   1:  PR[GP1:91,1] = PR[GP1:90,1] + 133.078;
   1:  PR[GP1:91,2] = PR[GP1:90,2] + 104.334;
   1:L PR[91] 10mm/sec FINE;
   1:  PR[GP1:91,1] = PR[GP1:90,1] + 132.574;
   1:  PR[GP1:91,2] = PR[GP1:90,2] + 104.937;
   1:L PR[91] 10mm/sec FINE;
   1:  PR[GP1:91,1] = PR[GP1:90,1] + 131.283;
   1:  PR[GP1:91,2] = PR[GP1:90,2] + 106.321;
   1:L PR[91] 10mm/sec FINE;
   1:  PR[GP1:91,1] = PR[GP1:90,1] + 130.348;
   1:  PR[GP1:91,2] = PR[GP1:90,2] + 107.265;
   1:L PR[91] 10mm/sec FINE;
   1:  PR[GP1:91,1] = PR[GP1:90,1] + 129.842;
   1:  PR[GP1:91,2] = PR[GP1:90,2] + 107.719;
   1:L PR[91] 10mm/sec FINE;
   1:  PR[GP1:91,1] = PR[GP1:90,1] + 128.720;
   1:  PR[GP1:91,2] = PR[GP1:90,2] + 108.706;
   1:L PR[91] 10mm/sec FINE;
   1:  PR[GP1:91,1] = PR[GP1:90,1] + 125.281;
   1:  PR[GP1:91,2] = PR[GP1:90,2] + 111.248;
   1:L PR[91] 10mm/sec FINE;
   1:  PR[GP1:91,1] = PR[GP1:90,1] + 124.815;
   1:  PR[GP1:91,2] = PR[GP1:90,2] + 111.519;
   1:L PR[91] 10mm/sec FINE;
   1:  PR[GP1:91,1] = PR[GP1:90,1] + 123.935;
   1:  PR[GP1:91,2] = PR[GP1:90,2] + 111.995;
   1:L PR[91] 10mm/sec FINE;
   1:  PR[GP1:91,1] = PR[GP1:90,1] + 122.852;
   1:  PR[GP1:91,2] = PR[GP1:90,2] + 112.673;
   1:L PR[91] 10mm/sec FINE;
   1:  PR[GP1:91,1] = PR[GP1:90,1] + 122.591;
   1:  PR[GP1:91,2] = PR[GP1:90,2] + 112.818;
   1:L PR[91] 10mm/sec FINE;
   1:  PR[GP1:91,1] = PR[GP1:90,1] + 122.383;
   1:  PR[GP1:91,2] = PR[GP1:90,2] + 112.910;
   1:L PR[91] 10mm/sec FINE;
   1:  PR[GP1:91,1] = PR[GP1:90,1] + 121.910;
   1:  PR[GP1:91,2] = PR[GP1:90,2] + 113.234;
   1:L PR[91] 10mm/sec FINE;
   1:  PR[GP1:91,1] = PR[GP1:90,1] + 120.972;
   1:  PR[GP1:91,2] = PR[GP1:90,2] + 113.697;
   1:L PR[91] 10mm/sec FINE;
   1:  PR[GP1:91,1] = PR[GP1:90,1] + 120.433;
   1:  PR[GP1:91,2] = PR[GP1:90,2] + 113.889;
   1:L PR[91] 10mm/sec FINE;
   1:  PR[GP1:91,1] = PR[GP1:90,1] + 118.110;
   1:  PR[GP1:91,2] = PR[GP1:90,2] + 115.002;
   1:L PR[91] 10mm/sec FINE;
   1:  PR[GP1:91,1] = PR[GP1:90,1] + 115.533;
   1:  PR[GP1:91,2] = PR[GP1:90,2] + 115.758;
   1:L PR[91] 10mm/sec FINE;
   1:  PR[GP1:91,1] = PR[GP1:90,1] + 114.209;
   1:  PR[GP1:91,2] = PR[GP1:90,2] + 116.169;
   1:L PR[91] 10mm/sec FINE;
   1:  PR[GP1:91,1] = PR[GP1:90,1] + 112.597;
   1:  PR[GP1:91,2] = PR[GP1:90,2] + 116.362;
   1:L PR[91] 10mm/sec FINE;
   1:  PR[GP1:91,1] = PR[GP1:90,1] + 110.291;
   1:  PR[GP1:91,2] = PR[GP1:90,2] + 116.663;
   1:L PR[91] 10mm/sec FINE;
   1:  PR[GP1:91,1] = PR[GP1:90,1] + 108.430;
   1:  PR[GP1:91,2] = PR[GP1:90,2] + 116.678;
   1:L PR[91] 10mm/sec FINE;
   1:  PR[GP1:91,1] = PR[GP1:90,1] + 104.683;
   1:  PR[GP1:91,2] = PR[GP1:90,2] + 116.533;
   1:L PR[91] 10mm/sec FINE;
   1:  PR[GP1:91,1] = PR[GP1:90,1] + 104.119;
   1:  PR[GP1:91,2] = PR[GP1:90,2] + 116.445;
   1:L PR[91] 10mm/sec FINE;
   1:  PR[GP1:91,1] = PR[GP1:90,1] + 100.824;
   1:  PR[GP1:91,2] = PR[GP1:90,2] + 115.784;
   1:L PR[91] 10mm/sec FINE;
   1:  PR[GP1:91,1] = PR[GP1:90,1] + 99.441;
   1:  PR[GP1:91,2] = PR[GP1:90,2] + 115.278;
   1:L PR[91] 10mm/sec FINE;
   1:  PR[GP1:91,1] = PR[GP1:90,1] + 97.150;
   1:  PR[GP1:91,2] = PR[GP1:90,2] + 114.379;
   1:L PR[91] 10mm/sec FINE;
   1:  PR[GP1:91,1] = PR[GP1:90,1] + 96.875;
   1:  PR[GP1:91,2] = PR[GP1:90,2] + 114.236;
   1:L PR[91] 10mm/sec FINE;
   1:  PR[GP1:91,1] = PR[GP1:90,1] + 94.091;
   1:  PR[GP1:91,2] = PR[GP1:90,2] + 112.451;
   1:L PR[91] 10mm/sec FINE;
   1:  PR[GP1:91,1] = PR[GP1:90,1] + 93.175;
   1:  PR[GP1:91,2] = PR[GP1:90,2] + 111.645;
   1:L PR[91] 10mm/sec FINE;
   1:  PR[GP1:91,1] = PR[GP1:90,1] + 91.727;
   1:  PR[GP1:91,2] = PR[GP1:90,2] + 110.082;
   1:L PR[91] 10mm/sec FINE;
   1:  PR[GP1:91,1] = PR[GP1:90,1] + 91.060;
   1:  PR[GP1:91,2] = PR[GP1:90,2] + 109.259;
   1:L PR[91] 10mm/sec FINE;
   1:  PR[GP1:91,1] = PR[GP1:90,1] + 90.553;
   1:  PR[GP1:91,2] = PR[GP1:90,2] + 108.353;
   1:L PR[91] 10mm/sec FINE;
   1:  PR[GP1:91,1] = PR[GP1:90,1] + 89.537;
   1:  PR[GP1:91,2] = PR[GP1:90,2] + 106.416;
   1:L PR[91] 10mm/sec FINE;
   1:  PR[GP1:91,1] = PR[GP1:90,1] + 89.209;
   1:  PR[GP1:91,2] = PR[GP1:90,2] + 105.500;
   1:L PR[91] 10mm/sec FINE;
   1:  PR[GP1:91,1] = PR[GP1:90,1] + 88.715;
   1:  PR[GP1:91,2] = PR[GP1:90,2] + 103.374;
   1:L PR[91] 10mm/sec FINE;
   1:  PR[GP1:91,1] = PR[GP1:90,1] + 88.529;
   1:  PR[GP1:91,2] = PR[GP1:90,2] + 102.358;
   1:L PR[91] 10mm/sec FINE;
   1:  PR[GP1:91,1] = PR[GP1:90,1] + 88.508;
   1:  PR[GP1:91,2] = PR[GP1:90,2] + 101.310;
   1:L PR[91] 10mm/sec FINE;
   1:  PR[GP1:91,1] = PR[GP1:90,1] + 88.621;
   1:  PR[GP1:91,2] = PR[GP1:90,2] + 99.170;
   1:L PR[91] 10mm/sec FINE;
   1:  PR[GP1:91,1] = PR[GP1:90,1] + 88.809;
   1:  PR[GP1:91,2] = PR[GP1:90,2] + 98.011;
   1:L PR[91] 10mm/sec FINE;
   1:  PR[GP1:91,1] = PR[GP1:90,1] + 88.822;
   1:  PR[GP1:91,2] = PR[GP1:90,2] + 97.961;
   1:L PR[91] 10mm/sec FINE;
   1:  PR[GP1:91,1] = PR[GP1:90,1] + 89.980;
   1:  PR[GP1:91,2] = PR[GP1:90,2] + 94.456;
   1:L PR[91] 10mm/sec FINE;
   1:  PR[GP1:91,1] = PR[GP1:90,1] + 90.236;
   1:  PR[GP1:91,2] = PR[GP1:90,2] + 93.612;
   1:L PR[91] 10mm/sec FINE;
   1:  PR[GP1:91,1] = PR[GP1:90,1] + 91.520;
   1:  PR[GP1:91,2] = PR[GP1:90,2] + 92.149;
   1:  PR[GP1:91,3] = PR[GP1:90,3] + 65.900;
   1:L PR[91] 10mm/sec FINE;
   1:  PR[GP1:91,1] = PR[GP1:90,1] + 92.735;
   1:  PR[GP1:91,2] = PR[GP1:90,2] + 90.111;
   1:L PR[91] 10mm/sec FINE;
   1:  PR[GP1:91,1] = PR[GP1:90,1] + 95.040;
   1:  PR[GP1:91,2] = PR[GP1:90,2] + 86.918;
   1:L PR[91] 10mm/sec FINE;
   1:  PR[GP1:91,1] = PR[GP1:90,1] + 96.371;
   1:  PR[GP1:91,2] = PR[GP1:90,2] + 85.475;
   1:L PR[91] 10mm/sec FINE;
   1:  PR[GP1:91,1] = PR[GP1:90,1] + 97.440;
   1:  PR[GP1:91,2] = PR[GP1:90,2] + 84.369;
   1:L PR[91] 10mm/sec FINE;
   1:  PR[GP1:91,1] = PR[GP1:90,1] + 101.784;
   1:  PR[GP1:91,2] = PR[GP1:90,2] + 80.978;
   1:L PR[91] 10mm/sec FINE;
   1:  PR[GP1:91,1] = PR[GP1:90,1] + 102.201;
   1:  PR[GP1:91,2] = PR[GP1:90,2] + 80.753;
   1:L PR[91] 10mm/sec FINE;
   1:  PR[GP1:91,1] = PR[GP1:90,1] + 106.860;
   1:  PR[GP1:91,2] = PR[GP1:90,2] + 78.023;
   1:L PR[91] 10mm/sec FINE;
   1:  PR[GP1:91,1] = PR[GP1:90,1] + 113.422;
   1:  PR[GP1:91,2] = PR[GP1:90,2] + 75.517;
   1:L PR[91] 10mm/sec FINE;
   1:  PR[GP1:91,1] = PR[GP1:90,1] + 117.856;
   1:  PR[GP1:91,2] = PR[GP1:90,2] + 74.650;
   1:L PR[91] 10mm/sec FINE;
   1:  PR[GP1:91,1] = PR[GP1:90,1] + 120.560;
   1:  PR[GP1:91,2] = PR[GP1:90,2] + 74.494;
   1:L PR[91] 10mm/sec FINE;
   1:  PR[GP1:91,1] = PR[GP1:90,1] + 121.439;
   1:  PR[GP1:91,2] = PR[GP1:90,2] + 74.463;
   1:L PR[91] 10mm/sec FINE;
   1:  PR[GP1:91,1] = PR[GP1:90,1] + 123.315;
   1:  PR[GP1:91,2] = PR[GP1:90,2] + 74.706;
   1:L PR[91] 10mm/sec FINE;
   1:  PR[GP1:91,1] = PR[GP1:90,1] + 125.689;
   1:  PR[GP1:91,2] = PR[GP1:90,2] + 74.966;
   1:L PR[91] 10mm/sec FINE;
   1:  PR[GP1:91,1] = PR[GP1:90,1] + 127.460;
   1:  PR[GP1:91,2] = PR[GP1:90,2] + 75.437;
   1:L PR[91] 10mm/sec FINE;
   1:  PR[GP1:91,1] = PR[GP1:90,1] + 130.068;
   1:  PR[GP1:91,2] = PR[GP1:90,2] + 76.445;
   1:L PR[91] 10mm/sec FINE;
   1:  PR[GP1:91,1] = PR[GP1:90,1] + 131.522;
   1:  PR[GP1:91,2] = PR[GP1:90,2] + 77.116;
   1:L PR[91] 10mm/sec FINE;
   1:  PR[GP1:91,1] = PR[GP1:90,1] + 132.509;
   1:  PR[GP1:91,2] = PR[GP1:90,2] + 77.819;
   1:L PR[91] 10mm/sec FINE;
   1:  PR[GP1:91,1] = PR[GP1:90,1] + 134.897;
   1:  PR[GP1:91,2] = PR[GP1:90,2] + 79.695;
   1:L PR[91] 10mm/sec FINE;
   1:  PR[GP1:91,1] = PR[GP1:90,1] + 135.682;
   1:  PR[GP1:91,2] = PR[GP1:90,2] + 80.533;
   1:L PR[91] 10mm/sec FINE;
   1:  PR[GP1:91,1] = PR[GP1:90,1] + 137.230;
   1:  PR[GP1:91,2] = PR[GP1:90,2] + 82.841;
   1:L PR[91] 10mm/sec FINE;
   1:  PR[GP1:91,1] = PR[GP1:90,1] + 137.802;
   1:  PR[GP1:91,2] = PR[GP1:90,2] + 83.791;
   1:L PR[91] 10mm/sec FINE;
   1:  PR[GP1:91,1] = PR[GP1:90,1] + 138.178;
   1:  PR[GP1:91,2] = PR[GP1:90,2] + 84.884;
   1:L PR[91] 10mm/sec FINE;
   1:  PR[GP1:91,1] = PR[GP1:90,1] + 138.856;
   1:  PR[GP1:91,2] = PR[GP1:90,2] + 86.970;
   1:L PR[91] 10mm/sec FINE;
   1:  PR[GP1:91,1] = PR[GP1:90,1] + 139.017;
   1:  PR[GP1:91,2] = PR[GP1:90,2] + 88.230;
   1:L PR[91] 10mm/sec FINE;
   1:  PR[GP1:91,1] = PR[GP1:90,1] + 139.191;
   1:  PR[GP1:91,2] = PR[GP1:90,2] + 90.045;
   1:L PR[91] 10mm/sec FINE;
   1:  PR[GP1:91,1] = PR[GP1:90,1] + 139.096;
   1:  PR[GP1:91,2] = PR[GP1:90,2] + 91.544;
   1:L PR[91] 10mm/sec FINE;
   1:  PR[GP1:91,1] = PR[GP1:90,1] + 138.958;
   1:  PR[GP1:91,2] = PR[GP1:90,2] + 93.171;
   1:L PR[91] 10mm/sec FINE;
   1:  PR[GP1:91,1] = PR[GP1:90,1] + 138.190;
   1:  PR[GP1:91,2] = PR[GP1:90,2] + 96.327;
   1:L PR[91] 10mm/sec FINE;
   1:  PR[GP1:91,1] = PR[GP1:90,1] + 137.095;
   1:  PR[GP1:91,2] = PR[GP1:90,2] + 99.086;
   1:L PR[91] 10mm/sec FINE;
   1:  PR[GP1:91,1] = PR[GP1:90,1] + 135.819;
   1:  PR[GP1:91,2] = PR[GP1:90,2] + 101.448;
   1:L PR[91] 10mm/sec FINE;
   1:  PR[GP1:91,1] = PR[GP1:90,1] + 135.643;
   1:  PR[GP1:91,2] = PR[GP1:90,2] + 101.737;
   1:L PR[91] 10mm/sec FINE;
   1:  PR[GP1:91,1] = PR[GP1:90,1] + 133.904;
   1:  PR[GP1:91,2] = PR[GP1:90,2] + 104.039;
   1:L PR[91] 10mm/sec FINE;
   1:  PR[GP1:91,1] = PR[GP1:90,1] + 133.599;
   1:  PR[GP1:91,2] = PR[GP1:90,2] + 104.403;
   1:L PR[91] 10mm/sec FINE;
   1:  PR[GP1:91,1] = PR[GP1:90,1] + 132.037;
   1:  PR[GP1:91,2] = PR[GP1:90,2] + 106.078;
   1:L PR[91] 10mm/sec FINE;
   1:  PR[GP1:91,1] = PR[GP1:90,1] + 131.332;
   1:  PR[GP1:91,2] = PR[GP1:90,2] + 106.790;
   1:L PR[91] 10mm/sec FINE;
   1:  PR[GP1:91,1] = PR[GP1:90,1] + 129.467;
   1:  PR[GP1:91,2] = PR[GP1:90,2] + 108.438;
   1:L PR[91] 10mm/sec FINE;
   1:  PR[GP1:91,1] = PR[GP1:90,1] + 127.205;
   1:  PR[GP1:91,2] = PR[GP1:90,2] + 110.116;
   1:L PR[91] 10mm/sec FINE;
   1:  PR[GP1:91,1] = PR[GP1:90,1] + 126.171;
   1:  PR[GP1:91,2] = PR[GP1:90,2] + 110.860;
   1:L PR[91] 10mm/sec FINE;
   1:  PR[GP1:91,1] = PR[GP1:90,1] + 125.079;
   1:  PR[GP1:91,2] = PR[GP1:90,2] + 111.497;
   1:L PR[91] 10mm/sec FINE;
   1:  PR[GP1:91,1] = PR[GP1:90,1] + 123.052;
   1:  PR[GP1:91,2] = PR[GP1:90,2] + 112.592;
   1:L PR[91] 10mm/sec FINE;
   1:  PR[GP1:91,1] = PR[GP1:90,1] + 122.515;
   1:  PR[GP1:91,2] = PR[GP1:90,2] + 112.928;
   1:L PR[91] 10mm/sec FINE;
   1:  PR[GP1:91,1] = PR[GP1:90,1] + 121.714;
   1:  PR[GP1:91,2] = PR[GP1:90,2] + 113.284;
   1:L PR[91] 10mm/sec FINE;
   1:  PR[GP1:91,1] = PR[GP1:90,1] + 120.818;
   1:  PR[GP1:91,2] = PR[GP1:90,2] + 113.730;
   1:L PR[91] 10mm/sec FINE;
   1:  PR[GP1:91,1] = PR[GP1:90,1] + 119.914;
   1:  PR[GP1:91,2] = PR[GP1:90,2] + 114.053;
   1:L PR[91] 10mm/sec FINE;
   1:  PR[GP1:91,1] = PR[GP1:90,1] + 118.581;
   1:  PR[GP1:91,2] = PR[GP1:90,2] + 114.689;
   1:L PR[91] 10mm/sec FINE;
   1:  PR[GP1:91,1] = PR[GP1:90,1] + 118.083;
   1:  PR[GP1:91,2] = PR[GP1:90,2] + 114.849;
   1:L PR[91] 10mm/sec FINE;
   1:  PR[GP1:91,1] = PR[GP1:90,1] + 117.577;
   1:  PR[GP1:91,2] = PR[GP1:90,2] + 114.961;
   1:L PR[91] 10mm/sec FINE;
   1:  PR[GP1:91,1] = PR[GP1:90,1] + 114.648;
   1:  PR[GP1:91,2] = PR[GP1:90,2] + 115.832;
   1:L PR[91] 10mm/sec FINE;
   1:  PR[GP1:91,1] = PR[GP1:90,1] + 110.715;
   1:  PR[GP1:91,2] = PR[GP1:90,2] + 116.315;
   1:L PR[91] 10mm/sec FINE;
   1:  PR[GP1:91,1] = PR[GP1:90,1] + 108.913;
   1:  PR[GP1:91,2] = PR[GP1:90,2] + 116.347;
   1:L PR[91] 10mm/sec FINE;
   1:  PR[GP1:91,1] = PR[GP1:90,1] + 105.317;
   1:  PR[GP1:91,2] = PR[GP1:90,2] + 116.207;
   1:L PR[91] 10mm/sec FINE;
   1:  PR[GP1:91,1] = PR[GP1:90,1] + 101.541;
   1:  PR[GP1:91,2] = PR[GP1:90,2] + 115.450;
   1:L PR[91] 10mm/sec FINE;
   1:  PR[GP1:91,1] = PR[GP1:90,1] + 100.669;
   1:  PR[GP1:91,2] = PR[GP1:90,2] + 115.131;
   1:L PR[91] 10mm/sec FINE;
   1:  PR[GP1:91,1] = PR[GP1:90,1] + 97.922;
   1:  PR[GP1:91,2] = PR[GP1:90,2] + 114.053;
   1:L PR[91] 10mm/sec FINE;
   1:  PR[GP1:91,1] = PR[GP1:90,1] + 97.589;
   1:  PR[GP1:91,2] = PR[GP1:90,2] + 113.880;
   1:L PR[91] 10mm/sec FINE;
   1:  PR[GP1:91,1] = PR[GP1:90,1] + 94.958;
   1:  PR[GP1:91,2] = PR[GP1:90,2] + 112.195;
   1:L PR[91] 10mm/sec FINE;
   1:  PR[GP1:91,1] = PR[GP1:90,1] + 93.796;
   1:  PR[GP1:91,2] = PR[GP1:90,2] + 111.173;
   1:L PR[91] 10mm/sec FINE;
   1:  PR[GP1:91,1] = PR[GP1:90,1] + 92.704;
   1:  PR[GP1:91,2] = PR[GP1:90,2] + 109.994;
   1:L PR[91] 10mm/sec FINE;
   1:  PR[GP1:91,1] = PR[GP1:90,1] + 91.816;
   1:  PR[GP1:91,2] = PR[GP1:90,2] + 108.898;
   1:L PR[91] 10mm/sec FINE;
   1:  PR[GP1:91,1] = PR[GP1:90,1] + 91.141;
   1:  PR[GP1:91,2] = PR[GP1:90,2] + 107.693;
   1:L PR[91] 10mm/sec FINE;
   1:  PR[GP1:91,1] = PR[GP1:90,1] + 90.375;
   1:  PR[GP1:91,2] = PR[GP1:90,2] + 106.232;
   1:L PR[91] 10mm/sec FINE;
   1:  PR[GP1:91,1] = PR[GP1:90,1] + 89.929;
   1:  PR[GP1:91,2] = PR[GP1:90,2] + 104.987;
   1:L PR[91] 10mm/sec FINE;
   1:  PR[GP1:91,1] = PR[GP1:90,1] + 89.557;
   1:  PR[GP1:91,2] = PR[GP1:90,2] + 103.384;
   1:L PR[91] 10mm/sec FINE;
   1:  PR[GP1:91,1] = PR[GP1:90,1] + 89.309;
   1:  PR[GP1:91,2] = PR[GP1:90,2] + 102.039;
   1:L PR[91] 10mm/sec FINE;
   1:  PR[GP1:91,1] = PR[GP1:90,1] + 89.283;
   1:  PR[GP1:91,2] = PR[GP1:90,2] + 100.651;
   1:L PR[91] 10mm/sec FINE;
   1:  PR[GP1:91,1] = PR[GP1:90,1] + 89.368;
   1:  PR[GP1:91,2] = PR[GP1:90,2] + 99.037;
   1:L PR[91] 10mm/sec FINE;
   1:  PR[GP1:91,1] = PR[GP1:90,1] + 89.522;
   1:  PR[GP1:91,2] = PR[GP1:90,2] + 98.084;
   1:L PR[91] 10mm/sec FINE;
   1:  PR[GP1:91,1] = PR[GP1:90,1] + 89.598;
   1:  PR[GP1:91,2] = PR[GP1:90,2] + 97.560;
   1:L PR[91] 10mm/sec FINE;
   1:  PR[GP1:91,1] = PR[GP1:90,1] + 90.483;
   1:  PR[GP1:91,2] = PR[GP1:90,2] + 94.868;
   1:L PR[91] 10mm/sec FINE;
   1:  PR[GP1:91,1] = PR[GP1:90,1] + 90.908;
   1:  PR[GP1:91,2] = PR[GP1:90,2] + 93.462;
   1:L PR[91] 10mm/sec FINE;
   1:  PR[GP1:91,1] = PR[GP1:90,1] + 92.439;
   1:  PR[GP1:91,2] = PR[GP1:90,2] + 91.470;
   1:  PR[GP1:91,3] = PR[GP1:90,3] + 66.900;
   1:L PR[91] 10mm/sec FINE;
   1:  PR[GP1:91,1] = PR[GP1:90,1] + 93.259;
   1:  PR[GP1:91,2] = PR[GP1:90,2] + 90.094;
   1:L PR[91] 10mm/sec FINE;
   1:  PR[GP1:91,1] = PR[GP1:90,1] + 96.052;
   1:  PR[GP1:91,2] = PR[GP1:90,2] + 86.224;
   1:L PR[91] 10mm/sec FINE;
   1:  PR[GP1:91,1] = PR[GP1:90,1] + 96.951;
   1:  PR[GP1:91,2] = PR[GP1:90,2] + 85.250;
   1:L PR[91] 10mm/sec FINE;
   1:  PR[GP1:91,1] = PR[GP1:90,1] + 98.166;
   1:  PR[GP1:91,2] = PR[GP1:90,2] + 83.993;
   1:L PR[91] 10mm/sec FINE;
   1:  PR[GP1:91,1] = PR[GP1:90,1] + 101.386;
   1:  PR[GP1:91,2] = PR[GP1:90,2] + 81.475;
   1:L PR[91] 10mm/sec FINE;
   1:  PR[GP1:91,1] = PR[GP1:90,1] + 102.269;
   1:  PR[GP1:91,2] = PR[GP1:90,2] + 80.719;
   1:L PR[91] 10mm/sec FINE;
   1:  PR[GP1:91,1] = PR[GP1:90,1] + 103.869;
   1:  PR[GP1:91,2] = PR[GP1:90,2] + 79.729;
   1:L PR[91] 10mm/sec FINE;
   1:  PR[GP1:91,1] = PR[GP1:90,1] + 107.640;
   1:  PR[GP1:91,2] = PR[GP1:90,2] + 77.520;
   1:L PR[91] 10mm/sec FINE;
   1:  PR[GP1:91,1] = PR[GP1:90,1] + 114.404;
   1:  PR[GP1:91,2] = PR[GP1:90,2] + 74.932;
   1:L PR[91] 10mm/sec FINE;
   1:  PR[GP1:91,1] = PR[GP1:90,1] + 118.646;
   1:  PR[GP1:91,2] = PR[GP1:90,2] + 74.108;
   1:L PR[91] 10mm/sec FINE;
   1:  PR[GP1:91,1] = PR[GP1:90,1] + 121.895;
   1:  PR[GP1:91,2] = PR[GP1:90,2] + 73.981;
   1:L PR[91] 10mm/sec FINE;
   1:  PR[GP1:91,1] = PR[GP1:90,1] + 123.161;
   1:  PR[GP1:91,2] = PR[GP1:90,2] + 74.146;
   1:L PR[91] 10mm/sec FINE;
   1:  PR[GP1:91,1] = PR[GP1:90,1] + 126.747;
   1:  PR[GP1:91,2] = PR[GP1:90,2] + 74.537;
   1:L PR[91] 10mm/sec FINE;
   1:  PR[GP1:91,1] = PR[GP1:90,1] + 127.938;
   1:  PR[GP1:91,2] = PR[GP1:90,2] + 74.854;
   1:L PR[91] 10mm/sec FINE;
   1:  PR[GP1:91,1] = PR[GP1:90,1] + 131.364;
   1:  PR[GP1:91,2] = PR[GP1:90,2] + 76.178;
   1:L PR[91] 10mm/sec FINE;
   1:  PR[GP1:91,1] = PR[GP1:90,1] + 132.341;
   1:  PR[GP1:91,2] = PR[GP1:90,2] + 76.629;
   1:L PR[91] 10mm/sec FINE;
   1:  PR[GP1:91,1] = PR[GP1:90,1] + 133.004;
   1:  PR[GP1:91,2] = PR[GP1:90,2] + 77.101;
   1:L PR[91] 10mm/sec FINE;
   1:  PR[GP1:91,1] = PR[GP1:90,1] + 135.886;
   1:  PR[GP1:91,2] = PR[GP1:90,2] + 79.365;
   1:L PR[91] 10mm/sec FINE;
   1:  PR[GP1:91,1] = PR[GP1:90,1] + 136.411;
   1:  PR[GP1:91,2] = PR[GP1:90,2] + 79.925;
   1:L PR[91] 10mm/sec FINE;
   1:  PR[GP1:91,1] = PR[GP1:90,1] + 138.258;
   1:  PR[GP1:91,2] = PR[GP1:90,2] + 82.679;
   1:L PR[91] 10mm/sec FINE;
   1:  PR[GP1:91,1] = PR[GP1:90,1] + 138.641;
   1:  PR[GP1:91,2] = PR[GP1:90,2] + 83.315;
   1:L PR[91] 10mm/sec FINE;
   1:  PR[GP1:91,1] = PR[GP1:90,1] + 138.893;
   1:  PR[GP1:91,2] = PR[GP1:90,2] + 84.049;
   1:L PR[91] 10mm/sec FINE;
   1:  PR[GP1:91,1] = PR[GP1:90,1] + 139.709;
   1:  PR[GP1:91,2] = PR[GP1:90,2] + 86.557;
   1:L PR[91] 10mm/sec FINE;
   1:  PR[GP1:91,1] = PR[GP1:90,1] + 139.816;
   1:  PR[GP1:91,2] = PR[GP1:90,2] + 87.404;
   1:L PR[91] 10mm/sec FINE;
   1:  PR[GP1:91,1] = PR[GP1:90,1] + 140.032;
   1:  PR[GP1:91,2] = PR[GP1:90,2] + 89.637;
   1:L PR[91] 10mm/sec FINE;
   1:  PR[GP1:91,1] = PR[GP1:90,1] + 139.968;
   1:  PR[GP1:91,2] = PR[GP1:90,2] + 90.647;
   1:L PR[91] 10mm/sec FINE;
   1:  PR[GP1:91,1] = PR[GP1:90,1] + 139.789;
   1:  PR[GP1:91,2] = PR[GP1:90,2] + 92.746;
   1:L PR[91] 10mm/sec FINE;
   1:  PR[GP1:91,1] = PR[GP1:90,1] + 139.029;
   1:  PR[GP1:91,2] = PR[GP1:90,2] + 95.851;
   1:L PR[91] 10mm/sec FINE;
   1:  PR[GP1:91,1] = PR[GP1:90,1] + 137.917;
   1:  PR[GP1:91,2] = PR[GP1:90,2] + 98.647;
   1:L PR[91] 10mm/sec FINE;
   1:  PR[GP1:91,1] = PR[GP1:90,1] + 136.476;
   1:  PR[GP1:91,2] = PR[GP1:90,2] + 101.303;
   1:L PR[91] 10mm/sec FINE;
   1:  PR[GP1:91,1] = PR[GP1:90,1] + 135.427;
   1:  PR[GP1:91,2] = PR[GP1:90,2] + 102.820;
   1:L PR[91] 10mm/sec FINE;
   1:  PR[GP1:91,1] = PR[GP1:90,1] + 134.621;
   1:  PR[GP1:91,2] = PR[GP1:90,2] + 103.873;
   1:L PR[91] 10mm/sec FINE;
   1:  PR[GP1:91,1] = PR[GP1:90,1] + 132.791;
   1:  PR[GP1:91,2] = PR[GP1:90,2] + 105.835;
   1:L PR[91] 10mm/sec FINE;
   1:  PR[GP1:91,1] = PR[GP1:90,1] + 132.315;
   1:  PR[GP1:91,2] = PR[GP1:90,2] + 106.315;
   1:L PR[91] 10mm/sec FINE;
   1:  PR[GP1:91,1] = PR[GP1:90,1] + 130.214;
   1:  PR[GP1:91,2] = PR[GP1:90,2] + 108.169;
   1:L PR[91] 10mm/sec FINE;
   1:  PR[GP1:91,1] = PR[GP1:90,1] + 128.684;
   1:  PR[GP1:91,2] = PR[GP1:90,2] + 109.303;
   1:L PR[91] 10mm/sec FINE;
   1:  PR[GP1:91,1] = PR[GP1:90,1] + 127.059;
   1:  PR[GP1:91,2] = PR[GP1:90,2] + 110.473;
   1:L PR[91] 10mm/sec FINE;
   1:  PR[GP1:91,1] = PR[GP1:90,1] + 125.343;
   1:  PR[GP1:91,2] = PR[GP1:90,2] + 111.474;
   1:L PR[91] 10mm/sec FINE;
   1:  PR[GP1:91,1] = PR[GP1:90,1] + 122.936;
   1:  PR[GP1:91,2] = PR[GP1:90,2] + 112.775;
   1:L PR[91] 10mm/sec FINE;
   1:  PR[GP1:91,1] = PR[GP1:90,1] + 122.527;
   1:  PR[GP1:91,2] = PR[GP1:90,2] + 112.964;
   1:L PR[91] 10mm/sec FINE;
   1:  PR[GP1:91,1] = PR[GP1:90,1] + 122.157;
   1:  PR[GP1:91,2] = PR[GP1:90,2] + 113.097;
   1:L PR[91] 10mm/sec FINE;
   1:  PR[GP1:91,1] = PR[GP1:90,1] + 121.062;
   1:  PR[GP1:91,2] = PR[GP1:90,2] + 113.543;
   1:L PR[91] 10mm/sec FINE;
   1:  PR[GP1:91,1] = PR[GP1:90,1] + 119.857;
   1:  PR[GP1:91,2] = PR[GP1:90,2] + 114.054;
   1:L PR[91] 10mm/sec FINE;
   1:  PR[GP1:91,1] = PR[GP1:90,1] + 119.395;
   1:  PR[GP1:91,2] = PR[GP1:90,2] + 114.216;
   1:L PR[91] 10mm/sec FINE;
   1:  PR[GP1:91,1] = PR[GP1:90,1] + 119.059;
   1:  PR[GP1:91,2] = PR[GP1:90,2] + 114.376;
   1:L PR[91] 10mm/sec FINE;
   1:  PR[GP1:91,1] = PR[GP1:90,1] + 117.912;
   1:  PR[GP1:91,2] = PR[GP1:90,2] + 114.745;
   1:L PR[91] 10mm/sec FINE;
   1:  PR[GP1:91,1] = PR[GP1:90,1] + 117.140;
   1:  PR[GP1:91,2] = PR[GP1:90,2] + 114.927;
   1:L PR[91] 10mm/sec FINE;
   1:  PR[GP1:91,1] = PR[GP1:90,1] + 116.777;
   1:  PR[GP1:91,2] = PR[GP1:90,2] + 114.996;
   1:L PR[91] 10mm/sec FINE;
   1:  PR[GP1:91,1] = PR[GP1:90,1] + 115.067;
   1:  PR[GP1:91,2] = PR[GP1:90,2] + 115.504;
   1:L PR[91] 10mm/sec FINE;
   1:  PR[GP1:91,1] = PR[GP1:90,1] + 114.243;
   1:  PR[GP1:91,2] = PR[GP1:90,2] + 115.630;
   1:L PR[91] 10mm/sec FINE;
   1:  PR[GP1:91,1] = PR[GP1:90,1] + 111.184;
   1:  PR[GP1:91,2] = PR[GP1:90,2] + 115.964;
   1:L PR[91] 10mm/sec FINE;
   1:  PR[GP1:91,1] = PR[GP1:90,1] + 111.102;
   1:  PR[GP1:91,2] = PR[GP1:90,2] + 115.968;
   1:L PR[91] 10mm/sec FINE;
   1:  PR[GP1:91,1] = PR[GP1:90,1] + 111.097;
   1:  PR[GP1:91,2] = PR[GP1:90,2] + 115.958;
   1:L PR[91] 10mm/sec FINE;
   1:  PR[GP1:91,1] = PR[GP1:90,1] + 109.881;
   1:  PR[GP1:91,2] = PR[GP1:90,2] + 116.011;
   1:L PR[91] 10mm/sec FINE;
   1:  PR[GP1:91,1] = PR[GP1:90,1] + 109.398;
   1:  PR[GP1:91,2] = PR[GP1:90,2] + 116.017;
   1:L PR[91] 10mm/sec FINE;
   1:  PR[GP1:91,1] = PR[GP1:90,1] + 106.940;
   1:  PR[GP1:91,2] = PR[GP1:90,2] + 115.924;
   1:L PR[91] 10mm/sec FINE;
   1:  PR[GP1:91,1] = PR[GP1:90,1] + 106.041;
   1:  PR[GP1:91,2] = PR[GP1:90,2] + 115.866;
   1:L PR[91] 10mm/sec FINE;
   1:  PR[GP1:91,1] = PR[GP1:90,1] + 102.257;
   1:  PR[GP1:91,2] = PR[GP1:90,2] + 115.115;
   1:L PR[91] 10mm/sec FINE;
   1:  PR[GP1:91,1] = PR[GP1:90,1] + 101.897;
   1:  PR[GP1:91,2] = PR[GP1:90,2] + 114.984;
   1:L PR[91] 10mm/sec FINE;
   1:  PR[GP1:91,1] = PR[GP1:90,1] + 98.694;
   1:  PR[GP1:91,2] = PR[GP1:90,2] + 113.727;
   1:L PR[91] 10mm/sec FINE;
   1:  PR[GP1:91,1] = PR[GP1:90,1] + 98.304;
   1:  PR[GP1:91,2] = PR[GP1:90,2] + 113.524;
   1:L PR[91] 10mm/sec FINE;
   1:  PR[GP1:91,1] = PR[GP1:90,1] + 95.824;
   1:  PR[GP1:91,2] = PR[GP1:90,2] + 111.938;
   1:L PR[91] 10mm/sec FINE;
   1:  PR[GP1:91,1] = PR[GP1:90,1] + 94.417;
   1:  PR[GP1:91,2] = PR[GP1:90,2] + 110.701;
   1:L PR[91] 10mm/sec FINE;
   1:  PR[GP1:91,1] = PR[GP1:90,1] + 93.681;
   1:  PR[GP1:91,2] = PR[GP1:90,2] + 109.907;
   1:L PR[91] 10mm/sec FINE;
   1:  PR[GP1:91,1] = PR[GP1:90,1] + 92.572;
   1:  PR[GP1:91,2] = PR[GP1:90,2] + 108.538;
   1:L PR[91] 10mm/sec FINE;
   1:  PR[GP1:91,1] = PR[GP1:90,1] + 91.729;
   1:  PR[GP1:91,2] = PR[GP1:90,2] + 107.032;
   1:L PR[91] 10mm/sec FINE;
   1:  PR[GP1:91,1] = PR[GP1:90,1] + 91.213;
   1:  PR[GP1:91,2] = PR[GP1:90,2] + 106.047;
   1:L PR[91] 10mm/sec FINE;
   1:  PR[GP1:91,1] = PR[GP1:90,1] + 90.649;
   1:  PR[GP1:91,2] = PR[GP1:90,2] + 104.475;
   1:L PR[91] 10mm/sec FINE;
   1:  PR[GP1:91,1] = PR[GP1:90,1] + 90.398;
   1:  PR[GP1:91,2] = PR[GP1:90,2] + 103.394;
   1:L PR[91] 10mm/sec FINE;
   1:  PR[GP1:91,1] = PR[GP1:90,1] + 90.090;
   1:  PR[GP1:91,2] = PR[GP1:90,2] + 101.720;
   1:L PR[91] 10mm/sec FINE;
   1:  PR[GP1:91,1] = PR[GP1:90,1] + 90.057;
   1:  PR[GP1:91,2] = PR[GP1:90,2] + 99.992;
   1:L PR[91] 10mm/sec FINE;
   1:  PR[GP1:91,1] = PR[GP1:90,1] + 90.114;
   1:  PR[GP1:91,2] = PR[GP1:90,2] + 98.905;
   1:L PR[91] 10mm/sec FINE;
   1:  PR[GP1:91,1] = PR[GP1:90,1] + 90.218;
   1:  PR[GP1:91,2] = PR[GP1:90,2] + 98.262;
   1:L PR[91] 10mm/sec FINE;
   1:  PR[GP1:91,1] = PR[GP1:90,1] + 90.387;
   1:  PR[GP1:91,2] = PR[GP1:90,2] + 97.099;
   1:L PR[91] 10mm/sec FINE;
   1:  PR[GP1:91,1] = PR[GP1:90,1] + 90.985;
   1:  PR[GP1:91,2] = PR[GP1:90,2] + 95.280;
   1:L PR[91] 10mm/sec FINE;
   1:  PR[GP1:91,1] = PR[GP1:90,1] + 91.581;
   1:  PR[GP1:91,2] = PR[GP1:90,2] + 93.312;
   1:L PR[91] 10mm/sec FINE;
   1:  PR[GP1:91,1] = PR[GP1:90,1] + 93.358;
   1:  PR[GP1:91,2] = PR[GP1:90,2] + 90.791;
   1:  PR[GP1:91,3] = PR[GP1:90,3] + 67.900;
   1:L PR[91] 10mm/sec FINE;
   1:  PR[GP1:91,1] = PR[GP1:90,1] + 93.783;
   1:  PR[GP1:91,2] = PR[GP1:90,2] + 90.078;
   1:L PR[91] 10mm/sec FINE;
   1:  PR[GP1:91,1] = PR[GP1:90,1] + 97.065;
   1:  PR[GP1:91,2] = PR[GP1:90,2] + 85.531;
   1:L PR[91] 10mm/sec FINE;
   1:  PR[GP1:91,1] = PR[GP1:90,1] + 97.531;
   1:  PR[GP1:91,2] = PR[GP1:90,2] + 85.025;
   1:L PR[91] 10mm/sec FINE;
   1:  PR[GP1:91,1] = PR[GP1:90,1] + 98.893;
   1:  PR[GP1:91,2] = PR[GP1:90,2] + 83.617;
   1:L PR[91] 10mm/sec FINE;
   1:  PR[GP1:91,1] = PR[GP1:90,1] + 100.576;
   1:  PR[GP1:91,2] = PR[GP1:90,2] + 82.300;
   1:L PR[91] 10mm/sec FINE;
   1:  PR[GP1:91,1] = PR[GP1:90,1] + 102.665;
   1:  PR[GP1:91,2] = PR[GP1:90,2] + 80.513;
   1:L PR[91] 10mm/sec FINE;
   1:  PR[GP1:91,1] = PR[GP1:90,1] + 106.452;
   1:  PR[GP1:91,2] = PR[GP1:90,2] + 78.169;
   1:L PR[91] 10mm/sec FINE;
   1:  PR[GP1:91,1] = PR[GP1:90,1] + 108.420;
   1:  PR[GP1:91,2] = PR[GP1:90,2] + 77.017;
   1:L PR[91] 10mm/sec FINE;
   1:  PR[GP1:91,1] = PR[GP1:90,1] + 115.387;
   1:  PR[GP1:91,2] = PR[GP1:90,2] + 74.347;
   1:L PR[91] 10mm/sec FINE;
   1:  PR[GP1:91,1] = PR[GP1:90,1] + 117.845;
   1:  PR[GP1:91,2] = PR[GP1:90,2] + 73.870;
   1:L PR[91] 10mm/sec FINE;
   1:  PR[GP1:91,1] = PR[GP1:90,1] + 120.493;
   1:  PR[GP1:91,2] = PR[GP1:90,2] + 73.565;
   1:L PR[91] 10mm/sec FINE;
   1:  PR[GP1:91,1] = PR[GP1:90,1] + 122.350;
   1:  PR[GP1:91,2] = PR[GP1:90,2] + 73.499;
   1:L PR[91] 10mm/sec FINE;
   1:  PR[GP1:91,1] = PR[GP1:90,1] + 123.007;
   1:  PR[GP1:91,2] = PR[GP1:90,2] + 73.585;
   1:L PR[91] 10mm/sec FINE;
   1:  PR[GP1:91,1] = PR[GP1:90,1] + 127.805;
   1:  PR[GP1:91,2] = PR[GP1:90,2] + 74.109;
   1:L PR[91] 10mm/sec FINE;
   1:  PR[GP1:91,1] = PR[GP1:90,1] + 128.417;
   1:  PR[GP1:91,2] = PR[GP1:90,2] + 74.272;
   1:L PR[91] 10mm/sec FINE;
   1:  PR[GP1:91,1] = PR[GP1:90,1] + 132.659;
   1:  PR[GP1:91,2] = PR[GP1:90,2] + 75.911;
   1:L PR[91] 10mm/sec FINE;
   1:  PR[GP1:91,1] = PR[GP1:90,1] + 133.160;
   1:  PR[GP1:91,2] = PR[GP1:90,2] + 76.142;
   1:L PR[91] 10mm/sec FINE;
   1:  PR[GP1:91,1] = PR[GP1:90,1] + 133.498;
   1:  PR[GP1:91,2] = PR[GP1:90,2] + 76.383;
   1:L PR[91] 10mm/sec FINE;
   1:  PR[GP1:91,1] = PR[GP1:90,1] + 136.875;
   1:  PR[GP1:91,2] = PR[GP1:90,2] + 79.036;
   1:L PR[91] 10mm/sec FINE;
   1:  PR[GP1:91,1] = PR[GP1:90,1] + 137.140;
   1:  PR[GP1:91,2] = PR[GP1:90,2] + 79.318;
   1:L PR[91] 10mm/sec FINE;
   1:  PR[GP1:91,1] = PR[GP1:90,1] + 139.285;
   1:  PR[GP1:91,2] = PR[GP1:90,2] + 82.517;
   1:L PR[91] 10mm/sec FINE;
   1:  PR[GP1:91,1] = PR[GP1:90,1] + 139.479;
   1:  PR[GP1:91,2] = PR[GP1:90,2] + 82.838;
   1:L PR[91] 10mm/sec FINE;
   1:  PR[GP1:91,1] = PR[GP1:90,1] + 140.561;
   1:  PR[GP1:91,2] = PR[GP1:90,2] + 86.145;
   1:L PR[91] 10mm/sec FINE;
   1:  PR[GP1:91,1] = PR[GP1:90,1] + 140.616;
   1:  PR[GP1:91,2] = PR[GP1:90,2] + 86.578;
   1:L PR[91] 10mm/sec FINE;
   1:  PR[GP1:91,1] = PR[GP1:90,1] + 140.872;
   1:  PR[GP1:91,2] = PR[GP1:90,2] + 89.230;
   1:L PR[91] 10mm/sec FINE;
   1:  PR[GP1:91,1] = PR[GP1:90,1] + 140.839;
   1:  PR[GP1:91,2] = PR[GP1:90,2] + 89.750;
   1:L PR[91] 10mm/sec FINE;
   1:  PR[GP1:91,1] = PR[GP1:90,1] + 140.620;
   1:  PR[GP1:91,2] = PR[GP1:90,2] + 92.320;
   1:L PR[91] 10mm/sec FINE;
   1:  PR[GP1:91,1] = PR[GP1:90,1] + 139.868;
   1:  PR[GP1:91,2] = PR[GP1:90,2] + 95.376;
   1:L PR[91] 10mm/sec FINE;
   1:  PR[GP1:91,1] = PR[GP1:90,1] + 138.739;
   1:  PR[GP1:91,2] = PR[GP1:90,2] + 98.207;
   1:L PR[91] 10mm/sec FINE;
   1:  PR[GP1:91,1] = PR[GP1:90,1] + 137.276;
   1:  PR[GP1:91,2] = PR[GP1:90,2] + 100.891;
   1:L PR[91] 10mm/sec FINE;
   1:  PR[GP1:91,1] = PR[GP1:90,1] + 136.035;
   1:  PR[GP1:91,2] = PR[GP1:90,2] + 102.686;
   1:L PR[91] 10mm/sec FINE;
   1:  PR[GP1:91,1] = PR[GP1:90,1] + 134.962;
   1:  PR[GP1:91,2] = PR[GP1:90,2] + 104.073;
   1:L PR[91] 10mm/sec FINE;
   1:  PR[GP1:91,1] = PR[GP1:90,1] + 133.297;
   1:  PR[GP1:91,2] = PR[GP1:90,2] + 105.842;
   1:L PR[91] 10mm/sec FINE;
   1:  PR[GP1:91,1] = PR[GP1:90,1] + 130.961;
   1:  PR[GP1:91,2] = PR[GP1:90,2] + 107.900;
   1:L PR[91] 10mm/sec FINE;
   1:  PR[GP1:91,1] = PR[GP1:90,1] + 130.164;
   1:  PR[GP1:91,2] = PR[GP1:90,2] + 108.491;
   1:L PR[91] 10mm/sec FINE;
   1:  PR[GP1:91,1] = PR[GP1:90,1] + 127.948;
   1:  PR[GP1:91,2] = PR[GP1:90,2] + 110.086;
   1:L PR[91] 10mm/sec FINE;
   1:  PR[GP1:91,1] = PR[GP1:90,1] + 125.606;
   1:  PR[GP1:91,2] = PR[GP1:90,2] + 111.452;
   1:L PR[91] 10mm/sec FINE;
   1:  PR[GP1:91,1] = PR[GP1:90,1] + 124.350;
   1:  PR[GP1:91,2] = PR[GP1:90,2] + 112.131;
   1:L PR[91] 10mm/sec FINE;
   1:  PR[GP1:91,1] = PR[GP1:90,1] + 122.657;
   1:  PR[GP1:91,2] = PR[GP1:90,2] + 112.915;
   1:L PR[91] 10mm/sec FINE;
   1:  PR[GP1:91,1] = PR[GP1:90,1] + 121.147;
   1:  PR[GP1:91,2] = PR[GP1:90,2] + 113.456;
   1:L PR[91] 10mm/sec FINE;
   1:  PR[GP1:91,1] = PR[GP1:90,1] + 119.601;
   1:  PR[GP1:91,2] = PR[GP1:90,2] + 114.086;
   1:L PR[91] 10mm/sec FINE;
   1:  PR[GP1:91,1] = PR[GP1:90,1] + 117.795;
   1:  PR[GP1:91,2] = PR[GP1:90,2] + 114.626;
   1:L PR[91] 10mm/sec FINE;
   1:  PR[GP1:91,1] = PR[GP1:90,1] + 117.573;
   1:  PR[GP1:91,2] = PR[GP1:90,2] + 114.681;
   1:L PR[91] 10mm/sec FINE;
   1:  PR[GP1:91,1] = PR[GP1:90,1] + 116.535;
   1:  PR[GP1:91,2] = PR[GP1:90,2] + 114.926;
   1:L PR[91] 10mm/sec FINE;
   1:  PR[GP1:91,1] = PR[GP1:90,1] + 115.975;
   1:  PR[GP1:91,2] = PR[GP1:90,2] + 115.032;
   1:L PR[91] 10mm/sec FINE;
   1:  PR[GP1:91,1] = PR[GP1:90,1] + 115.488;
   1:  PR[GP1:91,2] = PR[GP1:90,2] + 115.177;
   1:L PR[91] 10mm/sec FINE;
   1:  PR[GP1:91,1] = PR[GP1:90,1] + 113.764;
   1:  PR[GP1:91,2] = PR[GP1:90,2] + 115.439;
   1:L PR[91] 10mm/sec FINE;
   1:  PR[GP1:91,1] = PR[GP1:90,1] + 112.475;
   1:  PR[GP1:91,2] = PR[GP1:90,2] + 115.579;
   1:L PR[91] 10mm/sec FINE;
   1:  PR[GP1:91,1] = PR[GP1:90,1] + 109.904;
   1:  PR[GP1:91,2] = PR[GP1:90,2] + 115.686;
   1:L PR[91] 10mm/sec FINE;
   1:  PR[GP1:91,1] = PR[GP1:90,1] + 108.599;
   1:  PR[GP1:91,2] = PR[GP1:90,2] + 115.638;
   1:L PR[91] 10mm/sec FINE;
   1:  PR[GP1:91,1] = PR[GP1:90,1] + 106.736;
   1:  PR[GP1:91,2] = PR[GP1:90,2] + 115.518;
   1:L PR[91] 10mm/sec FINE;
   1:  PR[GP1:91,1] = PR[GP1:90,1] + 103.159;
   1:  PR[GP1:91,2] = PR[GP1:90,2] + 114.825;
   1:L PR[91] 10mm/sec FINE;
   1:  PR[GP1:91,1] = PR[GP1:90,1] + 102.679;
   1:  PR[GP1:91,2] = PR[GP1:90,2] + 114.677;
   1:L PR[91] 10mm/sec FINE;
   1:  PR[GP1:91,1] = PR[GP1:90,1] + 102.324;
   1:  PR[GP1:91,2] = PR[GP1:90,2] + 114.523;
   1:L PR[91] 10mm/sec FINE;
   1:  PR[GP1:91,1] = PR[GP1:90,1] + 99.467;
   1:  PR[GP1:91,2] = PR[GP1:90,2] + 113.402;
   1:L PR[91] 10mm/sec FINE;
   1:  PR[GP1:91,1] = PR[GP1:90,1] + 99.018;
   1:  PR[GP1:91,2] = PR[GP1:90,2] + 113.168;
   1:L PR[91] 10mm/sec FINE;
   1:  PR[GP1:91,1] = PR[GP1:90,1] + 96.690;
   1:  PR[GP1:91,2] = PR[GP1:90,2] + 111.682;
   1:L PR[91] 10mm/sec FINE;
   1:  PR[GP1:91,1] = PR[GP1:90,1] + 95.038;
   1:  PR[GP1:91,2] = PR[GP1:90,2] + 110.229;
   1:L PR[91] 10mm/sec FINE;
   1:  PR[GP1:91,1] = PR[GP1:90,1] + 94.658;
   1:  PR[GP1:91,2] = PR[GP1:90,2] + 109.819;
   1:L PR[91] 10mm/sec FINE;
   1:  PR[GP1:91,1] = PR[GP1:90,1] + 93.328;
   1:  PR[GP1:91,2] = PR[GP1:90,2] + 108.177;
   1:L PR[91] 10mm/sec FINE;
   1:  PR[GP1:91,1] = PR[GP1:90,1] + 92.318;
   1:  PR[GP1:91,2] = PR[GP1:90,2] + 106.372;
   1:L PR[91] 10mm/sec FINE;
   1:  PR[GP1:91,1] = PR[GP1:90,1] + 92.050;
   1:  PR[GP1:91,2] = PR[GP1:90,2] + 105.863;
   1:L PR[91] 10mm/sec FINE;
   1:  PR[GP1:91,1] = PR[GP1:90,1] + 91.369;
   1:  PR[GP1:91,2] = PR[GP1:90,2] + 103.962;
   1:L PR[91] 10mm/sec FINE;
   1:  PR[GP1:91,1] = PR[GP1:90,1] + 91.239;
   1:  PR[GP1:91,2] = PR[GP1:90,2] + 103.403;
   1:L PR[91] 10mm/sec FINE;
   1:  PR[GP1:91,1] = PR[GP1:90,1] + 90.871;
   1:  PR[GP1:91,2] = PR[GP1:90,2] + 101.401;
   1:L PR[91] 10mm/sec FINE;
   1:  PR[GP1:91,1] = PR[GP1:90,1] + 90.831;
   1:  PR[GP1:91,2] = PR[GP1:90,2] + 99.333;
   1:L PR[91] 10mm/sec FINE;
   1:  PR[GP1:91,1] = PR[GP1:90,1] + 90.861;
   1:  PR[GP1:91,2] = PR[GP1:90,2] + 98.772;
   1:L PR[91] 10mm/sec FINE;
   1:  PR[GP1:91,1] = PR[GP1:90,1] + 90.914;
   1:  PR[GP1:91,2] = PR[GP1:90,2] + 98.440;
   1:L PR[91] 10mm/sec FINE;
   1:  PR[GP1:91,1] = PR[GP1:90,1] + 91.176;
   1:  PR[GP1:91,2] = PR[GP1:90,2] + 96.638;
   1:L PR[91] 10mm/sec FINE;
   1:  PR[GP1:91,1] = PR[GP1:90,1] + 91.487;
   1:  PR[GP1:91,2] = PR[GP1:90,2] + 95.692;
   1:L PR[91] 10mm/sec FINE;
   1:  PR[GP1:91,1] = PR[GP1:90,1] + 92.253;
   1:  PR[GP1:91,2] = PR[GP1:90,2] + 93.163;
   1:L PR[91] 10mm/sec FINE;
   1:  PR[GP1:91,1] = PR[GP1:90,1] + 94.273;
   1:  PR[GP1:91,2] = PR[GP1:90,2] + 90.120;
   1:  PR[GP1:91,3] = PR[GP1:90,3] + 68.900;
   1:L PR[91] 10mm/sec FINE;
   1:  PR[GP1:91,1] = PR[GP1:90,1] + 98.076;
   1:  PR[GP1:91,2] = PR[GP1:90,2] + 84.839;
   1:L PR[91] 10mm/sec FINE;
   1:  PR[GP1:91,1] = PR[GP1:90,1] + 99.622;
   1:  PR[GP1:91,2] = PR[GP1:90,2] + 83.237;
   1:L PR[91] 10mm/sec FINE;
   1:  PR[GP1:91,1] = PR[GP1:90,1] + 103.062;
   1:  PR[GP1:91,2] = PR[GP1:90,2] + 80.307;
   1:L PR[91] 10mm/sec FINE;
   1:  PR[GP1:91,1] = PR[GP1:90,1] + 109.202;
   1:  PR[GP1:91,2] = PR[GP1:90,2] + 76.512;
   1:L PR[91] 10mm/sec FINE;
   1:  PR[GP1:91,1] = PR[GP1:90,1] + 116.369;
   1:  PR[GP1:91,2] = PR[GP1:90,2] + 73.762;
   1:L PR[91] 10mm/sec FINE;
   1:  PR[GP1:91,1] = PR[GP1:90,1] + 116.570;
   1:  PR[GP1:91,2] = PR[GP1:90,2] + 73.723;
   1:L PR[91] 10mm/sec FINE;
   1:  PR[GP1:91,1] = PR[GP1:90,1] + 122.659;
   1:  PR[GP1:91,2] = PR[GP1:90,2] + 73.023;
   1:L PR[91] 10mm/sec FINE;
   1:  PR[GP1:91,1] = PR[GP1:90,1] + 122.808;
   1:  PR[GP1:91,2] = PR[GP1:90,2] + 73.018;
   1:L PR[91] 10mm/sec FINE;
   1:  PR[GP1:91,1] = PR[GP1:90,1] + 128.853;
   1:  PR[GP1:91,2] = PR[GP1:90,2] + 73.679;
   1:L PR[91] 10mm/sec FINE;
   1:  PR[GP1:91,1] = PR[GP1:90,1] + 133.980;
   1:  PR[GP1:91,2] = PR[GP1:90,2] + 75.657;
   1:L PR[91] 10mm/sec FINE;
   1:  PR[GP1:91,1] = PR[GP1:90,1] + 137.877;
   1:  PR[GP1:91,2] = PR[GP1:90,2] + 78.723;
   1:L PR[91] 10mm/sec FINE;
   1:  PR[GP1:91,1] = PR[GP1:90,1] + 140.319;
   1:  PR[GP1:91,2] = PR[GP1:90,2] + 82.367;
   1:L PR[91] 10mm/sec FINE;
   1:  PR[GP1:91,1] = PR[GP1:90,1] + 141.413;
   1:  PR[GP1:91,2] = PR[GP1:90,2] + 85.729;
   1:L PR[91] 10mm/sec FINE;
   1:  PR[GP1:91,1] = PR[GP1:90,1] + 141.709;
   1:  PR[GP1:91,2] = PR[GP1:90,2] + 88.869;
   1:L PR[91] 10mm/sec FINE;
   1:  PR[GP1:91,1] = PR[GP1:90,1] + 141.451;
   1:  PR[GP1:91,2] = PR[GP1:90,2] + 91.895;
   1:L PR[91] 10mm/sec FINE;
   1:  PR[GP1:91,1] = PR[GP1:90,1] + 140.707;
   1:  PR[GP1:91,2] = PR[GP1:90,2] + 94.900;
   1:L PR[91] 10mm/sec FINE;
   1:  PR[GP1:91,1] = PR[GP1:90,1] + 139.561;
   1:  PR[GP1:91,2] = PR[GP1:90,2] + 97.768;
   1:L PR[91] 10mm/sec FINE;
   1:  PR[GP1:91,1] = PR[GP1:90,1] + 138.075;
   1:  PR[GP1:91,2] = PR[GP1:90,2] + 100.480;
   1:L PR[91] 10mm/sec FINE;
   1:  PR[GP1:91,1] = PR[GP1:90,1] + 137.971;
   1:  PR[GP1:91,2] = PR[GP1:90,2] + 100.631;
   1:L PR[91] 10mm/sec FINE;
   1:  PR[GP1:91,1] = PR[GP1:90,1] + 134.420;
   1:  PR[GP1:91,2] = PR[GP1:90,2] + 105.220;
   1:L PR[91] 10mm/sec FINE;
   1:  PR[GP1:91,1] = PR[GP1:90,1] + 134.281;
   1:  PR[GP1:91,2] = PR[GP1:90,2] + 105.368;
   1:L PR[91] 10mm/sec FINE;
   1:  PR[GP1:91,1] = PR[GP1:90,1] + 131.636;
   1:  PR[GP1:91,2] = PR[GP1:90,2] + 107.684;
   1:L PR[91] 10mm/sec FINE;
   1:  PR[GP1:91,1] = PR[GP1:90,1] + 128.836;
   1:  PR[GP1:91,2] = PR[GP1:90,2] + 109.699;
   1:L PR[91] 10mm/sec FINE;
   1:  PR[GP1:91,1] = PR[GP1:90,1] + 125.760;
   1:  PR[GP1:91,2] = PR[GP1:90,2] + 111.489;
   1:L PR[91] 10mm/sec FINE;
   1:  PR[GP1:91,1] = PR[GP1:90,1] + 122.787;
   1:  PR[GP1:91,2] = PR[GP1:90,2] + 112.865;
   1:L PR[91] 10mm/sec FINE;
   1:  PR[GP1:91,1] = PR[GP1:90,1] + 120.004;
   1:  PR[GP1:91,2] = PR[GP1:90,2] + 113.870;
   1:L PR[91] 10mm/sec FINE;
   1:  PR[GP1:91,1] = PR[GP1:90,1] + 119.504;
   1:  PR[GP1:91,2] = PR[GP1:90,2] + 114.022;
   1:L PR[91] 10mm/sec FINE;
   1:  PR[GP1:91,1] = PR[GP1:90,1] + 116.519;
   1:  PR[GP1:91,2] = PR[GP1:90,2] + 114.762;
   1:L PR[91] 10mm/sec FINE;
   1:  PR[GP1:91,1] = PR[GP1:90,1] + 113.352;
   1:  PR[GP1:91,2] = PR[GP1:90,2] + 115.227;
   1:L PR[91] 10mm/sec FINE;
   1:  PR[GP1:91,1] = PR[GP1:90,1] + 110.390;
   1:  PR[GP1:91,2] = PR[GP1:90,2] + 115.355;
   1:L PR[91] 10mm/sec FINE;
   1:  PR[GP1:91,1] = PR[GP1:90,1] + 107.431;
   1:  PR[GP1:91,2] = PR[GP1:90,2] + 115.171;
   1:L PR[91] 10mm/sec FINE;
   1:  PR[GP1:91,1] = PR[GP1:90,1] + 104.601;
   1:  PR[GP1:91,2] = PR[GP1:90,2] + 114.659;
   1:L PR[91] 10mm/sec FINE;
   1:  PR[GP1:91,1] = PR[GP1:90,1] + 102.218;
   1:  PR[GP1:91,2] = PR[GP1:90,2] + 113.928;
   1:L PR[91] 10mm/sec FINE;
   1:  PR[GP1:91,1] = PR[GP1:90,1] + 100.242;
   1:  PR[GP1:91,2] = PR[GP1:90,2] + 113.077;
   1:L PR[91] 10mm/sec FINE;
   1:  PR[GP1:91,1] = PR[GP1:90,1] + 99.733;
   1:  PR[GP1:91,2] = PR[GP1:90,2] + 112.812;
   1:L PR[91] 10mm/sec FINE;
   1:  PR[GP1:91,1] = PR[GP1:90,1] + 97.557;
   1:  PR[GP1:91,2] = PR[GP1:90,2] + 111.425;
   1:L PR[91] 10mm/sec FINE;
   1:  PR[GP1:91,1] = PR[GP1:90,1] + 95.629;
   1:  PR[GP1:91,2] = PR[GP1:90,2] + 109.723;
   1:L PR[91] 10mm/sec FINE;
   1:  PR[GP1:91,1] = PR[GP1:90,1] + 94.084;
   1:  PR[GP1:91,2] = PR[GP1:90,2] + 107.816;
   1:L PR[91] 10mm/sec FINE;
   1:  PR[GP1:91,1] = PR[GP1:90,1] + 92.887;
   1:  PR[GP1:91,2] = PR[GP1:90,2] + 105.676;
   1:L PR[91] 10mm/sec FINE;
   1:  PR[GP1:91,1] = PR[GP1:90,1] + 92.090;
   1:  PR[GP1:91,2] = PR[GP1:90,2] + 103.454;
   1:L PR[91] 10mm/sec FINE;
   1:  PR[GP1:91,1] = PR[GP1:90,1] + 91.652;
   1:  PR[GP1:91,2] = PR[GP1:90,2] + 101.082;
   1:L PR[91] 10mm/sec FINE;
   1:  PR[GP1:91,1] = PR[GP1:90,1] + 91.608;
   1:  PR[GP1:91,2] = PR[GP1:90,2] + 98.631;
   1:L PR[91] 10mm/sec FINE;
   1:  PR[GP1:91,1] = PR[GP1:90,1] + 91.965;
   1:  PR[GP1:91,2] = PR[GP1:90,2] + 96.178;
   1:L PR[91] 10mm/sec FINE;
   1:  PR[GP1:91,1] = PR[GP1:90,1] + 91.989;
   1:  PR[GP1:91,2] = PR[GP1:90,2] + 96.105;
   1:L PR[91] 10mm/sec FINE;
   1:  PR[GP1:91,1] = PR[GP1:90,1] + 92.925;
   1:  PR[GP1:91,2] = PR[GP1:90,2] + 93.013;
   1:L PR[91] 10mm/sec FINE;
   1:  PR[GP1:91,1] = PR[GP1:90,1] + 94.273;
   1:  PR[GP1:91,2] = PR[GP1:90,2] + 90.120;
   1:L PR[91] 10mm/sec FINE;
   1:  PR[GP1:91,1] = PR[GP1:90,1] + 98.076;
   1:  PR[GP1:91,2] = PR[GP1:90,2] + 84.839;
   1:L PR[91] 10mm/sec FINE;
   1:  PR[GP1:91,1] = PR[GP1:90,1] + 99.622;
   1:  PR[GP1:91,2] = PR[GP1:90,2] + 83.237;
   1:L PR[91] 10mm/sec FINE;
   1:  PR[GP1:91,1] = PR[GP1:90,1] + 103.062;
   1:  PR[GP1:91,2] = PR[GP1:90,2] + 80.307;
   1:L PR[91] 10mm/sec FINE;
   1:  PR[GP1:91,1] = PR[GP1:90,1] + 109.202;
   1:  PR[GP1:91,2] = PR[GP1:90,2] + 76.512;
   1:L PR[91] 10mm/sec FINE;
   1:  PR[GP1:91,1] = PR[GP1:90,1] + 116.369;
   1:  PR[GP1:91,2] = PR[GP1:90,2] + 73.762;
   1:L PR[91] 10mm/sec FINE;
   1:  PR[GP1:91,1] = PR[GP1:90,1] + 116.570;
   1:  PR[GP1:91,2] = PR[GP1:90,2] + 73.723;
   1:L PR[91] 10mm/sec FINE;
   1:  PR[GP1:91,1] = PR[GP1:90,1] + 122.659;
   1:  PR[GP1:91,2] = PR[GP1:90,2] + 73.023;
   1:L PR[91] 10mm/sec FINE;
   1:  PR[GP1:91,1] = PR[GP1:90,1] + 122.808;
   1:  PR[GP1:91,2] = PR[GP1:90,2] + 73.018;
   1:L PR[91] 10mm/sec FINE;
   1:  PR[GP1:91,1] = PR[GP1:90,1] + 128.853;
   1:  PR[GP1:91,2] = PR[GP1:90,2] + 73.679;
   1:L PR[91] 10mm/sec FINE;
   1:  PR[GP1:91,1] = PR[GP1:90,1] + 133.980;
   1:  PR[GP1:91,2] = PR[GP1:90,2] + 75.657;
   1:L PR[91] 10mm/sec FINE;
   1:  PR[GP1:91,1] = PR[GP1:90,1] + 137.877;
   1:  PR[GP1:91,2] = PR[GP1:90,2] + 78.723;
   1:L PR[91] 10mm/sec FINE;
   1:  PR[GP1:91,1] = PR[GP1:90,1] + 140.319;
   1:  PR[GP1:91,2] = PR[GP1:90,2] + 82.367;
   1:L PR[91] 10mm/sec FINE;
   1:  PR[GP1:91,1] = PR[GP1:90,1] + 141.413;
   1:  PR[GP1:91,2] = PR[GP1:90,2] + 85.729;
   1:L PR[91] 10mm/sec FINE;
   1:  PR[GP1:91,1] = PR[GP1:90,1] + 141.709;
   1:  PR[GP1:91,2] = PR[GP1:90,2] + 88.869;
   1:L PR[91] 10mm/sec FINE;
   1:  PR[GP1:91,1] = PR[GP1:90,1] + 141.451;
   1:  PR[GP1:91,2] = PR[GP1:90,2] + 91.895;
   1:L PR[91] 10mm/sec FINE;
   1:  PR[GP1:91,1] = PR[GP1:90,1] + 140.707;
   1:  PR[GP1:91,2] = PR[GP1:90,2] + 94.900;
   1:L PR[91] 10mm/sec FINE;
   1:  PR[GP1:91,1] = PR[GP1:90,1] + 139.561;
   1:  PR[GP1:91,2] = PR[GP1:90,2] + 97.768;
   1:L PR[91] 10mm/sec FINE;
   1:  PR[GP1:91,1] = PR[GP1:90,1] + 138.075;
   1:  PR[GP1:91,2] = PR[GP1:90,2] + 100.480;
   1:L PR[91] 10mm/sec FINE;
   1:  PR[GP1:91,1] = PR[GP1:90,1] + 137.971;
   1:  PR[GP1:91,2] = PR[GP1:90,2] + 100.631;
   1:L PR[91] 10mm/sec FINE;
   1:  PR[GP1:91,1] = PR[GP1:90,1] + 134.420;
   1:  PR[GP1:91,2] = PR[GP1:90,2] + 105.220;
   1:L PR[91] 10mm/sec FINE;
   1:  PR[GP1:91,1] = PR[GP1:90,1] + 134.281;
   1:  PR[GP1:91,2] = PR[GP1:90,2] + 105.368;
   1:L PR[91] 10mm/sec FINE;
   1:  PR[GP1:91,1] = PR[GP1:90,1] + 131.636;
   1:  PR[GP1:91,2] = PR[GP1:90,2] + 107.684;
   1:L PR[91] 10mm/sec FINE;
   1:  PR[GP1:91,1] = PR[GP1:90,1] + 128.836;
   1:  PR[GP1:91,2] = PR[GP1:90,2] + 109.699;
   1:L PR[91] 10mm/sec FINE;
   1:  PR[GP1:91,1] = PR[GP1:90,1] + 125.760;
   1:  PR[GP1:91,2] = PR[GP1:90,2] + 111.489;
   1:L PR[91] 10mm/sec FINE;
   1:  PR[GP1:91,1] = PR[GP1:90,1] + 122.787;
   1:  PR[GP1:91,2] = PR[GP1:90,2] + 112.865;
   1:L PR[91] 10mm/sec FINE;
   1:  PR[GP1:91,1] = PR[GP1:90,1] + 120.004;
   1:  PR[GP1:91,2] = PR[GP1:90,2] + 113.870;
   1:L PR[91] 10mm/sec FINE;
   1:  PR[GP1:91,1] = PR[GP1:90,1] + 119.504;
   1:  PR[GP1:91,2] = PR[GP1:90,2] + 114.022;
   1:L PR[91] 10mm/sec FINE;
   1:  PR[GP1:91,1] = PR[GP1:90,1] + 116.519;
   1:  PR[GP1:91,2] = PR[GP1:90,2] + 114.762;
   1:L PR[91] 10mm/sec FINE;
   1:  PR[GP1:91,1] = PR[GP1:90,1] + 113.352;
   1:  PR[GP1:91,2] = PR[GP1:90,2] + 115.227;
   1:L PR[91] 10mm/sec FINE;
   1:  PR[GP1:91,1] = PR[GP1:90,1] + 110.390;
   1:  PR[GP1:91,2] = PR[GP1:90,2] + 115.355;
   1:L PR[91] 10mm/sec FINE;
   1:  PR[GP1:91,1] = PR[GP1:90,1] + 107.431;
   1:  PR[GP1:91,2] = PR[GP1:90,2] + 115.171;
   1:L PR[91] 10mm/sec FINE;
   1:  PR[GP1:91,1] = PR[GP1:90,1] + 104.601;
   1:  PR[GP1:91,2] = PR[GP1:90,2] + 114.659;
   1:L PR[91] 10mm/sec FINE;
   1:  PR[GP1:91,1] = PR[GP1:90,1] + 102.218;
   1:  PR[GP1:91,2] = PR[GP1:90,2] + 113.928;
   1:L PR[91] 10mm/sec FINE;
   1:  PR[GP1:91,1] = PR[GP1:90,1] + 100.242;
   1:  PR[GP1:91,2] = PR[GP1:90,2] + 113.077;
   1:L PR[91] 10mm/sec FINE;
   1:  PR[GP1:91,1] = PR[GP1:90,1] + 99.733;
   1:  PR[GP1:91,2] = PR[GP1:90,2] + 112.812;
   1:L PR[91] 10mm/sec FINE;
   1:  PR[GP1:91,1] = PR[GP1:90,1] + 97.557;
   1:  PR[GP1:91,2] = PR[GP1:90,2] + 111.425;
   1:L PR[91] 10mm/sec FINE;
   1:  PR[GP1:91,1] = PR[GP1:90,1] + 95.629;
   1:  PR[GP1:91,2] = PR[GP1:90,2] + 109.723;
   1:L PR[91] 10mm/sec FINE;
   1:  PR[GP1:91,1] = PR[GP1:90,1] + 94.084;
   1:  PR[GP1:91,2] = PR[GP1:90,2] + 107.816;
   1:L PR[91] 10mm/sec FINE;
   1:  PR[GP1:91,1] = PR[GP1:90,1] + 92.887;
   1:  PR[GP1:91,2] = PR[GP1:90,2] + 105.676;
   1:L PR[91] 10mm/sec FINE;
   1:  PR[GP1:91,1] = PR[GP1:90,1] + 92.090;
   1:  PR[GP1:91,2] = PR[GP1:90,2] + 103.454;
   1:L PR[91] 10mm/sec FINE;
   1:  PR[GP1:91,1] = PR[GP1:90,1] + 91.652;
   1:  PR[GP1:91,2] = PR[GP1:90,2] + 101.082;
   1:L PR[91] 10mm/sec FINE;
   1:  PR[GP1:91,1] = PR[GP1:90,1] + 91.608;
   1:  PR[GP1:91,2] = PR[GP1:90,2] + 98.631;
   1:L PR[91] 10mm/sec FINE;
   1:  PR[GP1:91,1] = PR[GP1:90,1] + 91.965;
   1:  PR[GP1:91,2] = PR[GP1:90,2] + 96.178;
   1:L PR[91] 10mm/sec FINE;
   1:  PR[GP1:91,1] = PR[GP1:90,1] + 91.989;
   1:  PR[GP1:91,2] = PR[GP1:90,2] + 96.105;
   1:L PR[91] 10mm/sec FINE;
   1:  PR[GP1:91,1] = PR[GP1:90,1] + 92.925;
   1:  PR[GP1:91,2] = PR[GP1:90,2] + 93.013;
   1:L PR[91] 10mm/sec FINE;
   1:  CALL HOME_ALL;
/POS
/END
